(* Logix 5000 project; controller EWEB_SOCK_TCP_SERV_VER2_1 1756-L62 rev 15.4; software revision 15.02 *)

TASK MainTask (periodic, rate 5 ms, priority 10, watchdog 500 ms) : MainProgram

MODULES
   Local : 1756-L62 (ICP 4, rev 15.4)
END_MODULES

TYPE AcceptResponse :
STRUCT
   Instance : DINT;
   Addr : SockAddr;
END_STRUCT
END_TYPE

TYPE OpenConnParam :
STRUCT
   Timeout : DINT;
   DestAddr : STRING;
END_STRUCT
END_TYPE

TYPE READ_DATA_REQ :
STRUCT
   Timeout : DINT;
   BufLen : DINT;
END_STRUCT
END_TYPE

TYPE READ_RESP :
STRUCT
   FromAddr : SockAddr;
   READ_BUFF : STR_4096;
END_STRUCT
END_TYPE

TYPE REQUEST_PARAMETERS :
STRUCT
   Type : DINT;   // 1 - TCP 2- UPD
   Addr : SockAddr;
END_STRUCT
END_TYPE

TYPE SockAddr :
STRUCT
   Family : INT;   // Address Family Must be 2
   Port : INT;   // Port Number
   Addr : DINT;   // IP Address
END_STRUCT
END_TYPE

TYPE STR_4096 :
STRUCT
   LEN : DINT;
   DATA : SINT[4096];
END_STRUCT
END_TYPE

TYPE STR_480 :
STRUCT
   LEN : DINT;
   DATA : SINT[480];
END_STRUCT
END_TYPE

TYPE Write_Data :
STRUCT
   Timeout : DINT;
   ToAddr : SockAddr;
   BufLen : DINT;
   Buf : SINT[20];
END_STRUCT
END_TYPE

TYPE WRT_DATA :
STRUCT
   Timeout : DINT;
   ToAddr : SockAddr;
   Buffer : STR_480;
END_STRUCT
END_TYPE

VAR_GLOBAL   (* controller tags *)
   _EWEB_PATH : STRING := '$01$07';
   Accept : ALIAS FOR Log_Enable.2;
   Accept_Request : BOOL;   // Toggle this Bit to Accept Incoming Connection
   Attrubute : ALIAS FOR Log_Enable.6;
   BufLenSent : DINT := 7;
   Change_Log_Msg : MESSAGE;
        MessageParameters(ServiceCode := 16#0010, LocalElement := Log_Enable, ...)
   CLOCK : DINT[7] := ([0] := 1998, [1] := 1, [2] := 12, [3] := 22, [4] := 11, [5] := 13, [6] := 576094);
   COLN : STRING := ':';
   Conn_Accept_MSG : MESSAGE;
        MessageParameters(ServiceCode := 16#0050, LocalElement := Sock_Accept_Timeout, DestinationTag := Sock_Accept_Resp, ...)
   Create : ALIAS FOR Log_Enable.0;
   Create_Sock_MSG : MESSAGE;
        MessageParameters(ServiceCode := 16#004b, LocalElement := Socket, DestinationTag := Instance, ...)
   Create_Socket_Req : BOOL;
   Delete : ALIAS FOR Log_Enable.5;
   Delete_All_MSG : MESSAGE;
        MessageParameters(ServiceCode := 16#0051, ...)
   Delete_All_Request : BOOL;
   Delete_Sock_MSG : MESSAGE;
        MessageParameters(ServiceCode := 16#004f, ...)
   Delete_Sockets_Req : BOOL;
   Enable_Log_MSG : MESSAGE;
        MessageParameters(ServiceCode := 16#000e, DestinationTag := Log_Enable, ...)
   Enable_Log_Req : BOOL;
   Errors : ALIAS FOR Log_Enable.7;
   Get_Sock_Instance_MSG : MESSAGE;
        MessageParameters(ServiceCode := 16#0001, DestinationTag := Sock_Object_Data[0], ...)
   Get_Sock_Object_MSG : MESSAGE;
        MessageParameters(ServiceCode := 16#0001, DestinationTag := Socket_Object_Class_Response[0], ...)
   Get_Socket_Instance_Req : BOOL;
   Get_Socket_Object_Req : BOOL;
   HOUR : STRING := '22';
   Instance : DINT := 484;
   Log_Enable : DINT := 255;
   Log_old : DINT;
   MINUTE : STRING := '11';
   Nothing : BOOL := 1;
   Open : ALIAS FOR Log_Enable.1;
   Read : ALIAS FOR Log_Enable.3;
   Read_Data_MSG : MESSAGE;
        MessageParameters(ServiceCode := 16#004d, LocalElement := Read_Data_Req, DestinationTag := Read_Response, ...)
   Read_Data_Req : READ_DATA_REQ := (Timeout := 1000, BufLen := 100);
   Read_Data_Request : BOOL;   // Toggle This Bit to Read Incoming Data
   Read_Response : READ_RESP := (READ_BUFF := '07:50:1207:50:1307:50:14');
   SECOND : STRING := '13';
   Sock_Accept_Resp : AcceptResponse := (Instance := 4805, Addr.Family := 2, Addr.Port := 1188, Addr.Addr := 1684298241);
   Sock_Accept_Timeout : DINT := 26000;
   Sock_Object_Data : DINT[13] := ([0] := 655425538, [4] := 2048, [5] := 2048, [6] := 8, [7] := 1, [8] := 300000);
   Socket : REQUEST_PARAMETERS := (Type := 1, Addr.Family := 2, Addr.Port := 10002);
   Socket_Object_Class_Response : SINT[10] := ([0] := 1, [2] := 20);
   TIME : STRING := '22:11:13';
   Write : ALIAS FOR Log_Enable.4;
   Write_Data_MSG : MESSAGE;
        MessageParameters(ServiceCode := 16#004e, LocalElement := Write_Data_Out, DestinationTag := BufLenSent, ...)
   Write_Data_Out : WRT_DATA := (Timeout := 20000, ToAddr.Family := 2, Buffer := '22:11:13');
   Write_Request : BOOL;   // Toggle This Bit to Send Data Out
   zero : STRING := '0';
END_VAR

PROGRAM MainProgram   (* main routine _SOCKET_TCP_SERV *)

ROUTINE _SOCKET_STATS   (* ladder *)
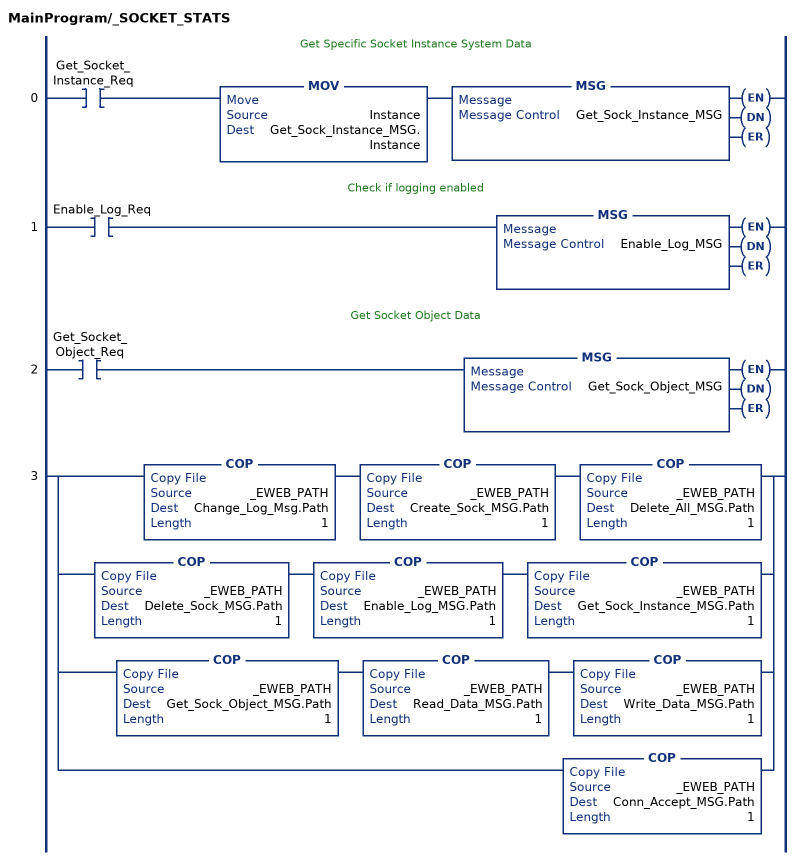
   // Get Specific Socket Instance System Data
   0: XIC(Get_Socket_Instance_Req)MOV(Instance,Get_Sock_Instance_MSG.Instance)MSG(Get_Sock_Instance_MSG);
   // Check if logging enabled
   1: XIC(Enable_Log_Req)MSG(Enable_Log_MSG);
   // Get Socket Object Data
   2: XIC(Get_Socket_Object_Req)MSG(Get_Sock_Object_MSG);
   3: [COP(_EWEB_PATH,Change_Log_Msg.Path,1) COP(_EWEB_PATH,Create_Sock_MSG.Path,1) COP(_EWEB_PATH,Delete_All_MSG.Path,1) ,COP(_EWEB_PATH,Delete_Sock_MSG.Path,1) COP(_EWEB_PATH,Enable_Log_MSG.Path,1) COP(_EWEB_PATH,Get_Sock_Instance_MSG.Path,1) ,COP(_EWEB_PATH,Get_Sock_Object_MSG.Path,1) COP(_EWEB_PATH,Read_Data_MSG.Path,1) COP(_EWEB_PATH,Write_Data_MSG.Path,1) ,COP(_EWEB_PATH,Conn_Accept_MSG.Path,1) ];
END_ROUTINE

ROUTINE _SOCKET_TCP_SERV   (* ladder *)
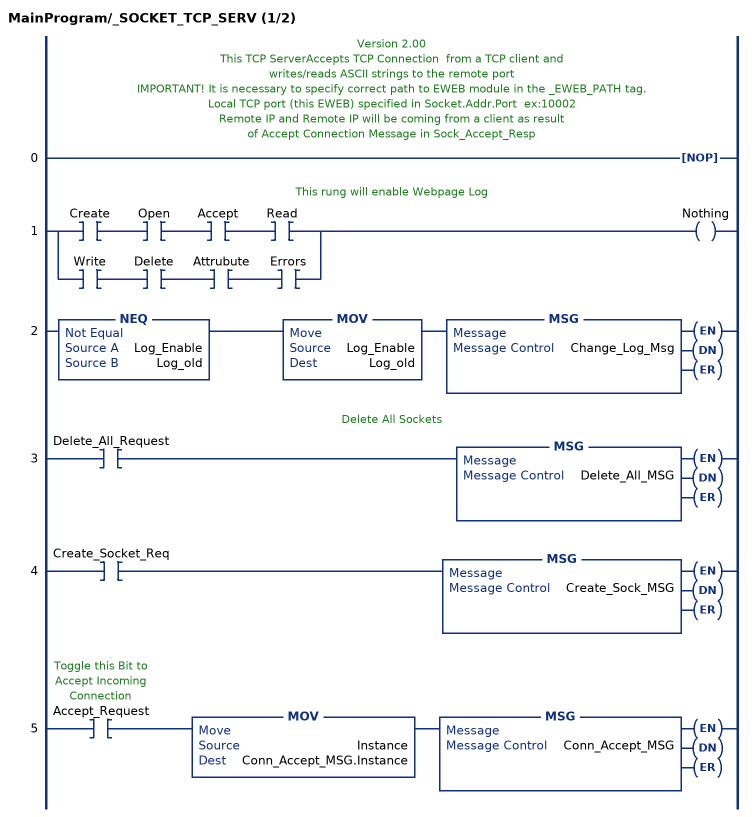
   // Version 2.00
   // This TCP ServerAccepts TCP Connection  from a TCP client and
   // writes/reads ASCII strings to the remote port
   // IMPORTANT! It is necessary to specify correct path to EWEB module in the _EWEB_PATH tag.
   // Local TCP port (this EWEB) specified in Socket.Addr.Port  ex:10002
   // Remote IP and Remote IP will be coming from a client as result
   // of Accept Connection Message in Sock_Accept_Resp
   0: NOP();
   // This rung will enable Webpage Log
   1: [XIC(Create) XIC(Open) XIC(Accept) XIC(Read) ,XIC(Write) XIC(Delete) XIC(Attrubute) XIC(Errors) ]OTE(Nothing);
   2: NEQ(Log_Enable,Log_old)MOV(Log_Enable,Log_old)MSG(Change_Log_Msg);
   // Delete All Sockets
   3: XIC(Delete_All_Request)MSG(Delete_All_MSG);
   4: XIC(Create_Socket_Req)MSG(Create_Sock_MSG);
   5: XIC(Accept_Request)MOV(Instance,Conn_Accept_MSG.Instance)MSG(Conn_Accept_MSG);
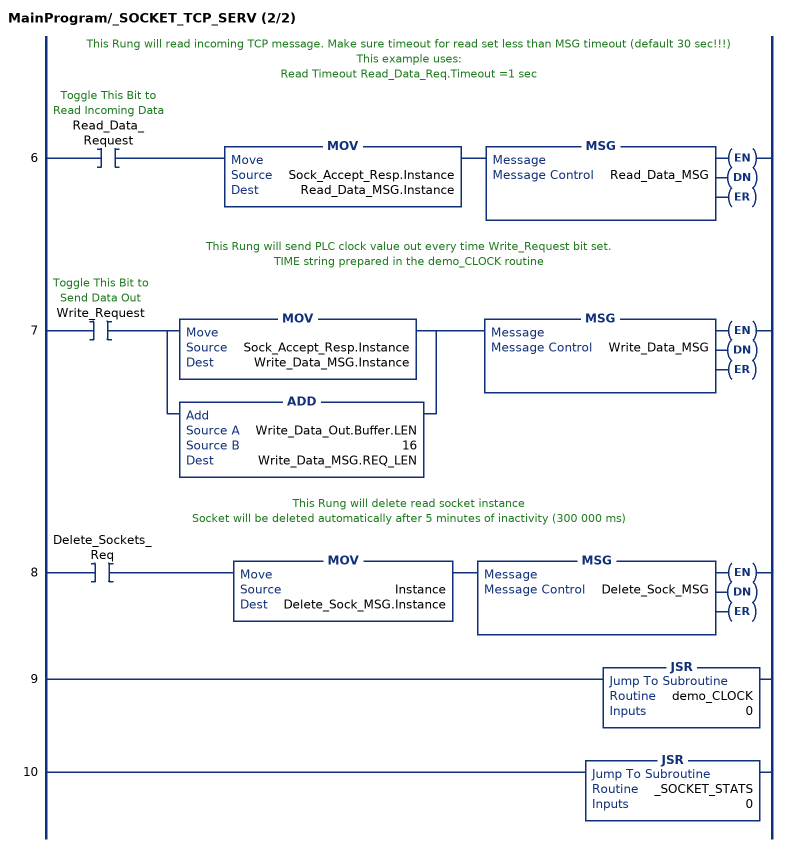
   // This Rung will read incoming TCP message. Make sure timeout for read set less than MSG timeout (default 30 sec!!!)
   // This example uses:
   // Read Timeout Read_Data_Req.Timeout =1 sec
   6: XIC(Read_Data_Request)MOV(Sock_Accept_Resp.Instance,Read_Data_MSG.Instance)MSG(Read_Data_MSG);
   // This Rung will send PLC clock value out every time Write_Request bit set.
   // TIME string prepared in the demo_CLOCK routine
   7: XIC(Write_Request)[MOV(Sock_Accept_Resp.Instance,Write_Data_MSG.Instance) ,ADD(Write_Data_Out.Buffer.LEN,16,Write_Data_MSG.REQ_LEN) ]MSG(Write_Data_MSG);
   // This Rung will delete read socket instance
   // Socket will be deleted automatically after 5 minutes of inactivity (300 000 ms)
   8: XIC(Delete_Sockets_Req)MOV(Instance,Delete_Sock_MSG.Instance)MSG(Delete_Sock_MSG);
   9: JSR(demo_CLOCK,0);
   10: JSR(_SOCKET_STATS,0);
END_ROUTINE

ROUTINE demo_CLOCK   (* ladder *)
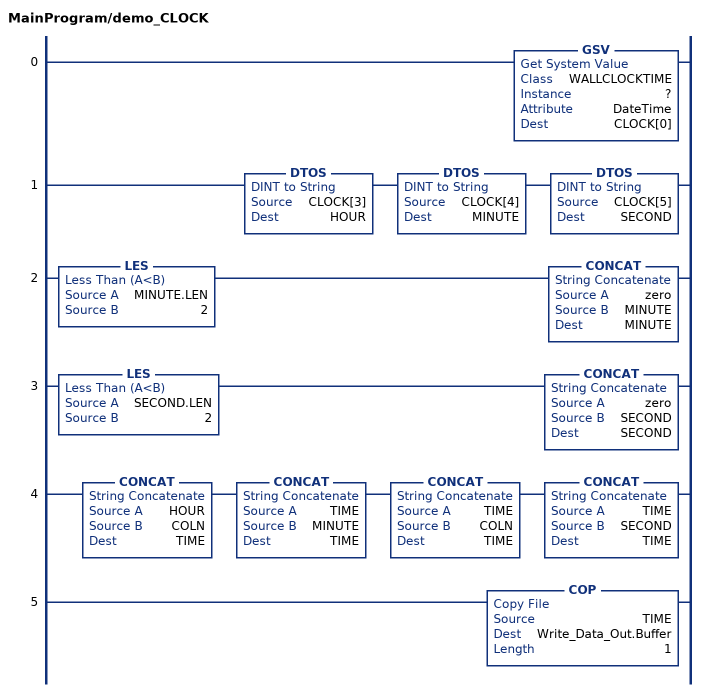
   0: GSV(WALLCLOCKTIME,?,DateTime,CLOCK[0]);
   1: DTOS(CLOCK[3],HOUR)DTOS(CLOCK[4],MINUTE)DTOS(CLOCK[5],SECOND);
   2: LES(MINUTE.LEN,2)CONCAT(zero,MINUTE,MINUTE);
   3: LES(SECOND.LEN,2)CONCAT(zero,SECOND,SECOND);
   4: CONCAT(HOUR,COLN,TIME)CONCAT(TIME,MINUTE,TIME)CONCAT(TIME,COLN,TIME)CONCAT(TIME,SECOND,TIME);
   5: COP(TIME,Write_Data_Out.Buffer,1);
END_ROUTINE
END_PROGRAM
